Yaskawa INFORM job: FMTV_FENDERS.JBI

/JOB
//NAME FMTV_FENDERS
//POS
///NPOS 545,0,0,3,0,0
///TOOL 0
///POSTYPE PULSE
///PULSE
C00000=-63956,-155148,126845,-105314,-81595,-126672
C00001=-236501,-175042,15743,-102650,-110361,-51662
C00002=-236501,-175042,-85215,-102650,-110361,-73822
C00003=-248122,-122895,-115006,-97112,-80000,-47589
C00004=-248635,-127033,-112745,-102549,-53011,-48741
C00005=-234079,-137705,-95028,-87046,-41878,-79782
C00006=-238942,-134708,-94740,-89961,-45016,-68159
C00007=-242508,-132671,-97164,-92994,-47428,-52176
C00008=-224790,-161630,-99096,-61743,-42779,-71567
C00009=-225833,-166497,-100724,-75197,-37378,-66529
C00010=-225972,-169847,-101473,-88583,-33472,-60957
C00011=-240574,-167077,-99779,-106864,-55530,-59132
C00012=-246383,-162026,-96863,-119993,-73009,-60358
C00013=-241063,-171089,-91582,-115750,-67016,-71356
C00014=-234594,-170823,-91883,-123396,-77107,-68502
C00015=-231990,-170973,-91438,-122280,-75787,-65647
C00016=-218685,-173595,-93676,-116936,-69568,-59454
C00017=-209410,-168993,-95200,-117606,-79816,-56023
C00018=-205376,-166532,-94796,-118730,-93657,-54826
C00019=-205520,-167299,-149545,-118775,-93902,539
C00020=194752,-167299,-149545,-204519,-57378,33957
C00021=227777,-146515,-121429,-211592,-64921,47742
C00022=140813,-165782,-97540,-184911,-23121,3391
C00023=142401,-166246,-97145,-186466,-22763,-397
C00024=129538,-168092,-98000,-174243,-22289,-10940
C00025=108353,-169637,-101483,-151757,-24269,-29279
C00026=76493,-168015,-109892,-143048,-39020,-42938
C00027=71930,-167798,-152447,-142497,-39770,-44912
C00028=-184184,-167798,-152447,-142497,-39770,-44912
C00029=-188241,-175091,-112594,-105313,-81595,-75530
C00030=-137238,-129578,-121502,-201786,-71124,-123955
C00031=-113155,-108086,-93765,-247340,-66179,-146822
C00032=-87884,-87482,-101015,-240031,-88214,-149958
C00033=-87337,-86742,-96838,-237644,-87662,-149095
C00034=-86639,-91328,-99206,-236722,-87486,-148429
C00035=-86780,-92686,-99571,-236735,-87113,-148223
C00036=-87673,-96396,-100101,-236785,-85664,-145021
C00037=-90528,-100864,-97206,-241818,-78899,-142882
C00038=-88930,-100173,-90592,-254807,-82341,-140248
C00039=-88930,-100173,-90592,-254807,-82341,-140248
C00040=-91958,-101268,-92449,-250564,-79276,-141210
C00041=-93563,-102238,-93369,-248531,-77706,-141653
C00042=-119301,-108319,-88132,-240089,-57325,-143963
C00043=-119660,-108541,-87987,-240161,-57013,-143942
C00044=-119839,-108971,-88005,-240265,-56797,-143863
C00045=-120234,-109926,-88726,-240307,-56496,-143882
C00046=-121927,-111036,-90334,-239348,-55531,-144622
C00047=-118976,-116509,-91716,-240930,-60604,-142515
C00048=-116081,-121406,-92670,-241702,-65588,-140629
C00049=-113168,-125880,-93367,-241813,-70447,-138887
C00050=-109736,-130380,-93806,-241238,-75765,-137011
C00051=-105270,-135511,-94001,-239583,-82236,-134673
C00052=-98930,-140934,-93505,-236003,-90100,-131558
C00053=-89867,-146515,-92095,-228369,-100341,-126955
C00054=-89580,-147813,-92127,-228164,-100030,-126621
C00055=-90841,-147991,-91556,-228656,-99205,-126757
C00056=-96418,-152558,-96101,-230948,-96589,-127979
C00057=-91724,-166412,-117528,-260601,-98993,-131473
C00058=-142876,-156018,-103642,-277845,-66892,-131209
C00059=-141572,-151863,-98523,-277546,-67748,-131008
C00060=-143622,-155846,-98171,-279282,-66778,-129574
C00061=-141572,-151863,-98523,-277546,-67748,-131008
C00062=-172590,-143236,-94657,-288827,-48166,-129963
C00063=-191755,-131411,-90127,-295423,-35245,-129238
C00064=-192589,-130434,-90093,-295337,-34548,-129452
C00065=-191324,-128508,-89233,-293789,-35094,-130268
C00066=-170465,-108298,-84931,-276180,-46986,-139791
C00067=-170465,-108298,-84931,-276180,-46986,-139791
C00068=-170175,-107085,-84636,-275676,-47146,-140161
C00069=-170577,-105937,-83925,-275538,-46851,-140322
C00070=-169650,-103921,-80673,-282063,-48979,-138868
C00071=-168642,-102219,-80355,-281188,-49540,-139276
C00072=-169071,-108002,-93409,-278198,-48715,-141830
C00073=-169071,-108002,-93409,-278198,-48715,-141830
C00074=-47220,-130234,-115451,-278198,-65852,-141829
C00075=198695,-175103,-103633,-278198,-100436,-141828
C00076=239511,-167652,-97207,-278198,-100438,-141828
C00077=238443,-174672,23867,-278198,-100438,-141828
C00078=2947,-175103,38446,-278198,-100436,-36834
C00079=16726,-130618,77154,-263150,-91818,-20452
C00080=23551,-123817,76415,-256358,-86647,-25076
C00081=25255,-134753,53984,-254887,-87968,-28104
C00082=34217,-129882,61937,-248584,-86650,-23141
C00083=34992,-129505,62675,-248048,-86512,-23065
C00084=35569,-128900,63365,-247642,-86445,-23063
C00085=35569,-128900,63365,-247642,-86445,-23063
C00086=35569,-128900,63365,-247642,-86445,-23063
C00087=35799,-128709,63623,-247480,-86412,-23052
C00088=36324,-128461,64149,-247118,-86309,-22994
C00089=36692,-142226,36581,-233091,-77214,-27321
C00090=36971,-139485,43358,-233271,-75982,-27198
C00091=42868,-132233,61112,-235070,-77346,-25322
C00092=50739,-147582,43443,-222735,-62053,-31597
C00093=47831,-140548,57273,-230647,-62785,-28767
C00094=34340,-130815,75810,-246275,-65428,-24880
C00095=33507,-162796,67711,-252752,-61051,-17702
C00096=33260,-171150,47504,-183611,-66896,-17832
C00097=100012,-174561,95289,18814,-62607,-57140
C00098=99763,-174577,58172,18619,-63102,-57088
C00099=101096,-171100,56758,19675,-60596,-57340
C00100=84534,-174582,50021,23554,-70995,-76849
C00101=83318,-171811,53916,22816,-71627,-76924
C00102=83719,-170735,55890,22980,-71982,-76759
C00103=84083,-169443,57369,23169,-72011,-76683
C00104=82602,-172191,48669,33395,-63575,-78747
C00105=81200,-174768,38987,47055,-54860,-82592
C00106=83526,-167021,50934,46962,-56546,-75402
C00107=83546,-144153,93765,41175,-74852,-61002
C00108=81875,-142151,96395,45526,-72096,-57806
C00109=83151,-130904,116355,41565,-65822,-44019
C00110=83644,-126633,124240,39180,-65180,-40041
C00111=83534,-127495,122450,39269,-64858,-40238
C00112=84956,-132447,112751,40602,-62697,-40874
C00113=87573,-136499,104656,41438,-60781,-40939
C00114=89464,-137800,101703,41543,-59955,-40657
C00115=90888,-139642,97462,43059,-58642,-40845
C00116=92923,-141988,91755,45353,-56827,-41168
C00117=97347,-145437,82552,50313,-53590,-41778
C00118=101127,-147299,76883,54509,-51347,-42234
C00119=112694,-149561,67089,67207,-46322,-43420
C00120=112404,-142486,73485,67419,-46217,-43743
C00121=112249,-142557,71998,67965,-45978,-44258
C00122=112309,-135857,81532,66813,-46484,-43309
C00123=112423,-127896,93799,65107,-47307,-41879
C00124=112481,-118724,108063,63143,-48368,-40240
C00125=112694,-149561,67089,67207,-46322,-43420
C00126=112694,-149561,67089,67207,-46322,-43420
C00127=116026,-148180,67774,69460,-45423,-43446
C00128=118687,-144460,72072,70778,-44893,-43092
C00129=113027,-132465,87179,66269,-46758,-27490
C00130=113284,-132594,85154,67245,-46318,-28134
C00131=117715,-137204,78104,70883,-44882,-37107
C00132=118231,-136060,79389,71132,-44786,-37034
C00133=118721,-135959,79407,71463,-44662,-37033
C00134=139669,-145382,63973,87795,-39566,-47806
C00135=144694,-152917,52086,93827,-38613,-57145
C00136=151618,-163514,32928,104061,-38168,-72003
C00137=153104,-166256,24026,108879,-38853,-74649
C00138=149828,-162760,31507,104102,-38640,-63057
C00139=147298,-159676,37324,100611,-38673,-54667
C00140=147603,-160409,36248,101031,-38660,-54816
C00141=147925,-161389,34936,101456,-38648,-54956
C00142=148129,-162398,33663,101755,-38646,-55064
C00143=147893,-163417,32335,102136,-38757,-54575
C00144=146258,-164194,31781,100421,-38883,-51526
C00145=140568,-164282,32355,94404,-49003,-49367
C00146=133209,-162489,36110,88716,-64281,-46826
C00147=128857,-160624,39192,86775,-74962,-45374
C00148=126945,-159418,41079,86406,-80510,-44608
C00149=124614,-158041,43286,86500,-87890,-43559
C00150=124939,-153213,57755,86544,-88151,-40924
C00151=125394,-169115,39061,86896,-87980,-41582
C00152=125574,-175038,-5981,87026,-114787,-41677
C00153=125574,-175038,-98531,87026,-114787,-41677
C00154=-224301,-140149,-112569,-110141,-97352,-69368
C00155=-229663,-142484,-108537,-111899,-99628,-71764
C00156=-230892,-138053,-104282,-112208,-100447,-71858
C00157=-228508,-142108,-101165,-112055,-97629,-73428
C00158=-230003,-144530,-99119,-112804,-97681,-74805
C00159=-237315,-146893,-98401,-115581,-101333,-76663
C00160=-237192,-144365,-100145,-122189,-107894,-76884
C00161=-235565,-140992,-101778,-130482,-115488,-77678
C00162=-235563,-141001,-101786,-130481,-115487,-77677
C00163=-237825,-141777,-101649,-131712,-116315,-78485
C00164=-238364,-143167,-100756,-132394,-115806,-79161
C00165=-226999,-153783,-87557,-130027,-102586,-81819
C00166=-222820,-155853,-86813,-128215,-99812,-81611
C00167=-216816,-162804,-92469,-125449,-96634,-80821
C00168=-216816,-162804,-92469,-125449,-96634,-80821
C00169=50184,-164124,-141814,36356,38768,-145446
C00170=54442,-155394,-111475,22539,120746,-180496
C00171=51486,-150306,-107537,20755,122050,-181495
C00172=63426,-151628,-102258,27464,115883,-177940
C00173=71735,-149481,-97078,31867,112002,-175642
C00174=81923,-149105,-93748,36922,107221,-173076
C00175=93853,-150952,-94431,42518,102084,-170079
C00176=97845,-151639,-92939,44162,99620,-169505
C00177=100339,-151371,-92202,45229,98399,-168996
C00178=100309,-151030,-92216,45235,98542,-168932
C00179=100415,-149962,-92546,45356,98998,-168621
C00180=111889,-132617,-94399,56113,85553,-159405
C00181=116128,-123385,-93936,57705,78449,-155514
C00182=119709,-114359,-92766,57352,71837,-151949
C00183=122591,-105709,-90679,55611,66072,-148743
C00184=121430,-103362,-88798,55594,66891,-148891
C00185=120850,-102704,-88701,55530,67390,-148888
C00186=120281,-102346,-88871,55475,67872,-148893
C00187=103719,-103787,-98738,55205,79854,-156387
C00188=103861,-103141,-98570,55164,79915,-156243
C00189=96021,-102003,-100562,55140,85368,-157297
C00190=90958,-101699,-103793,55098,89327,-157636
C00191=89909,-100879,-104523,55097,90388,-157513
C00192=89807,-100027,-104366,55100,90656,-157377
C00193=89221,-98801,-103895,56224,91516,-157316
C00194=88766,-97677,-103297,57173,92190,-157270
C00195=89816,-94344,-102182,57192,92197,-156513
C00196=96964,-101233,-114771,56885,89487,-153707
C00197=96964,-175067,-154909,56885,89487,-153707
C00198=-188147,-175067,-154909,56885,89487,-153707
C00199=-249562,-175082,-16518,56885,115648,-153706
C00200=-188145,-175086,16419,56885,121874,-153706
C00201=-177417,-173959,29423,-34415,105748,-147371
C00202=-215218,-169631,-6124,-67662,97554,-158481
C00203=-212851,-170254,-11358,-66279,98657,-160355
C00204=-199538,-170974,-5542,-56389,98010,-158467
C00205=-196518,-171702,4598,-68884,91761,-156498
C00206=-191507,-170789,17376,-83691,87075,-153205
C00207=-184847,-169628,24159,-91154,83928,-151061
C00208=-184769,-168513,30877,-91403,83962,-149508
C00209=-166653,-153882,67375,-118564,90914,-139805
C00210=-168376,-157673,56992,-119714,89739,-141501
C00211=-170268,-156203,59245,-123438,80532,-141325
C00212=-171412,-154267,62166,-126915,71162,-140836
C00213=-171531,-154006,62478,-127383,69855,-140765
C00214=-172026,-152514,64166,-129774,63219,-140319
C00215=-172277,-150476,66358,-132476,56004,-139609
C00216=-172404,-145153,73532,-132977,56608,-139199
C00217=-171743,-142696,76210,-132662,56537,-139081
C00218=-175468,-149312,61635,-117570,52509,-146387
C00219=-182053,-156892,41178,-91409,54589,-159429
C00220=-179598,-153809,48467,-91200,54250,-158022
C00221=-177876,-151695,51361,-90271,53969,-157773
C00222=-175031,-149700,54466,-88701,53470,-157416
C00223=-171138,-149200,55226,-90700,51887,-155676
C00224=-152905,-141663,70200,-105827,48301,-143509
C00225=-152337,-141979,69626,-105360,48147,-143575
C00226=-151943,-142781,68394,-104935,48012,-143705
C00227=-148029,-134110,86517,-121166,52616,-135065
C00228=-146834,-130705,93327,-125465,54888,-132704
C00229=-145103,-124844,104734,-130953,58789,-129572
C00230=-142768,-113260,126814,-137507,65892,-125434
C00231=-135917,-118098,122435,-150990,58780,-120039
C00232=-136643,-115604,126770,-151681,59833,-118172
C00233=-133945,-127048,108732,-147879,54997,-122652
C00234=-132685,-131473,101421,-146007,52903,-123186
C00235=-131275,-135352,94587,-143913,50769,-123796
C00236=-131275,-135352,94587,-143913,50769,-123796
C00237=-131275,-135352,94587,-143913,50769,-123796
C00238=-121206,-145281,78428,-130981,41887,-126182
C00239=-108596,-150086,71319,-118128,35191,-127801
C00240=-108596,-150086,71319,-118128,35191,-127801
C00241=-108596,-150086,71319,-118128,35191,-127801
C00242=-106173,-149311,73486,-117873,34909,-126912
C00243=-105014,-148827,74616,-117745,34762,-126490
C00244=-103301,-148028,76337,-117552,34523,-125880
C00245=-101267,-148049,76425,-114785,33084,-126447
C00246=-98887,-147633,77014,-111606,31465,-127110
C00247=-99861,-135336,105011,-122576,35238,-120303
C00248=-79582,-141041,101392,-54417,-60770,-149548
C00249=-78156,-144611,92640,-54931,-59723,-148027
C00250=-76477,-145690,87146,-55172,-58933,-146653
C00251=-76325,-152698,75551,-53287,-65768,-134624
C00252=-76716,-159478,64431,-47040,-68901,-125086
C00253=-79518,-161789,63221,-35636,-69401,-124582
C00254=-81209,-163290,61958,-29327,-69264,-124632
C00255=-84722,-166411,58236,-19438,-67363,-126288
C00256=-86671,-168300,55657,-13814,-66439,-127558
C00257=-86671,-168300,55657,-13814,-66439,-127558
C00258=-86216,-169741,53857,-13592,-66313,-127456
C00259=-85119,-170597,52676,-13583,-66937,-127129
C00260=-82515,-161498,64875,-12910,-80387,-133971
C00261=-77611,-145974,86579,-16344,-98063,-141066
C00262=-78076,-150431,78979,-16594,-96561,-139590
C00263=-80411,-152118,77648,-18159,-96529,-140021
C00264=-82668,-153005,77611,-19681,-96705,-140485
C00265=-88888,-175086,79531,-19379,-96436,-140350
C00266=-110968,-175086,9069,-19379,-125140,-140350
C00267=-110968,-175086,-114864,-19379,-125140,-140350
C00268=175304,-175086,-114864,-19379,-30472,-99694
C00269=187329,-129396,-122749,-38461,29346,-63021
C00270=183916,-109052,-100373,-57748,65750,-30233
C00271=197239,-90135,-82008,-58535,73988,-27553
C00272=201754,-94869,-83954,-58993,75937,-25896
C00273=202079,-95139,-84115,-59008,76103,-25800
C00274=202637,-95511,-84460,-59016,76432,-25674
C00275=202637,-95511,-84460,-59016,76432,-25674
C00276=202637,-95511,-84460,-59016,76432,-25674
C00277=202860,-95637,-84608,-59016,76571,-25633
C00278=203690,-96180,-85102,-59023,77053,-25445
C00279=208915,-99439,-88258,-58000,79285,-28016
C00280=205478,-105010,-93814,-58035,77197,-28705
C00281=214139,-97501,-89593,-72382,81942,-36081
C00282=224242,-84526,-78845,-86787,78269,-51115
C00283=224432,-83745,-74911,-87107,78310,-50227
C00284=223676,-86642,-76315,-87324,77734,-49801
C00285=223812,-88001,-76982,-87395,77808,-49593
C00286=224543,-88686,-77346,-87375,78313,-49481
C00287=235420,-107309,-83637,-91467,63449,-46681
C00288=240320,-114099,-85995,-93455,57854,-45609
C00289=246996,-121668,-88445,-96053,51244,-44273
C00290=246996,-121668,-88445,-96053,51244,-44273
C00291=249717,-122652,-88778,-95572,53097,-44156
C00292=250120,-123785,-89127,-95767,53405,-43893
C00293=232812,-141826,-96443,-115069,24978,-36767
C00294=232812,-141826,-96443,-115069,24978,-36767
C00295=233391,-143923,-96937,-116153,25668,-36002
C00296=237215,-145543,-97234,-114188,28169,-36484
C00297=245415,-146262,-97619,-108727,33105,-38331
C00298=245415,-146262,-97619,-108727,33105,-38331
C00299=247668,-147105,-97798,-107850,34572,-38441
C00300=248141,-148229,-98044,-108198,34996,-38104
C00301=248169,-149917,-101541,-106958,34753,-38928
C00302=248344,-161240,-125557,-97827,33569,-44956
C00303=179896,-161240,-125557,-97827,-77291,-48113
C00304=184979,-139013,-125331,-99817,-75478,-48047
C00305=179112,-130483,-99577,-98597,-78190,-53181
C00306=178361,-129263,-96461,-98549,-78560,-53744
C00307=161550,-139106,-101847,-102031,-89241,-56097
C00308=150835,-139809,-97057,-95903,-96892,-60596
C00309=132439,-136388,-86127,-87364,-112558,-64828
C00310=125150,-133069,-79774,-83061,-119517,-65455
C00311=123583,-134542,-82111,-83279,-120436,-65117
C00312=123583,-134540,-118710,-83279,-120438,-65115
C00313=-136821,-161457,-114880,15988,-123554,-94299
C00314=-194311,-175100,-121530,66302,-125133,-109092
C00315=-194311,-175100,-121530,-44006,100681,-109092
C00316=-254343,-175097,-89612,-83602,114959,-15902
C00317=-134289,-173861,-75426,-80327,116995,-14503
C00318=-122808,-169798,-71461,-73331,121943,-13820
C00319=-204100,-166260,-61655,-119208,88598,-10349
C00320=-223955,-164817,-61952,-125089,83393,-8296
C00321=-234599,-164424,-61970,-128682,80581,-6975
C00322=-239551,-164319,-62025,-130691,79207,-6317
C00323=-239846,-164373,-60068,-133976,79268,-5541
C00324=-241352,-164565,-58325,-139265,78932,-4470
C00325=-241352,-164565,-58325,-139265,78932,-4470
C00326=-241352,-164565,-58325,-139265,78932,-4470
C00327=-247260,-164414,-57679,-143144,77614,-3349
C00328=-250453,-164099,-56779,-145288,77091,-2673
C00329=-231804,-169514,-49324,-147051,71343,-6571
C00330=-232933,-169740,-48497,-147965,71587,-6225
C00331=-232886,-175090,-53650,-147961,71735,-6180
C00332=-241976,-170697,-124750,-139782,79456,-4031
C00333=-176745,-151691,-107508,-102764,25310,-35154
C00334=-176745,-151691,-107508,-102764,25310,-35154
C00335=-175824,-150531,-104417,-104152,26105,-34141
C00336=-176745,-151691,-107508,-102764,25310,-35154
C00337=-195718,-137133,-102300,-100933,12070,-39089
C00338=-195586,-136734,-99661,-105865,12408,-36294
C00339=-195718,-137133,-102300,-100933,12070,-39089
C00340=-180125,-124233,-99711,-80430,22769,-49034
C00341=-179992,-123952,-97169,-83121,22691,-47416
C00342=-180125,-124233,-99711,-80430,22769,-49034
C00343=-162775,-136432,-106392,-85396,34185,-43914
C00344=-162116,-135482,-103340,-86834,34551,-42863
C00345=-162775,-136432,-106392,-85396,34185,-43914
C00346=-136686,-149350,-103002,-109734,61122,-29919
C00347=-106697,-140430,-78975,-133534,56483,-36128
C00348=-113088,-137327,-73738,-138383,54551,-33834
C00349=-113904,-135440,-73782,-138477,53489,-34041
C00350=-109003,-138587,-73014,-136035,56934,-34530
C00351=-120827,-140923,-75250,-144601,52532,-30939
C00352=-120374,-136814,-75228,-143259,51004,-31973
C00353=-120840,-133958,-75226,-142869,49667,-32458
C00354=-120840,-133958,-75226,-142869,49667,-32458
C00355=-118039,-132206,-74509,-140437,50317,-33657
C00356=-114795,-132712,-73740,-138398,52103,-34407
C00357=-113063,-135707,-73613,-137984,53990,-34190
C00358=-109736,-137390,-76478,-135398,54956,-35431
C00359=-89018,-147818,-96006,-121054,62352,-42706
C00360=-127918,-122489,-87741,-140529,17400,-4354
C00361=-127917,-122488,-87741,-140529,17399,-4355
C00362=-120737,-122510,-87236,-129675,21028,-9702
C00363=-118823,-120927,-84702,-128126,22316,-10351
C00364=-119175,-120684,-84537,-128485,22104,-10188
C00365=-118541,-120339,-84470,-127414,22352,-10732
C00366=-117917,-120545,-84643,-126699,22698,-11070
C00367=-117746,-121573,-84792,-127367,23061,-10647
C00368=-117746,-121573,-84792,-127367,23061,-10647
C00369=-118346,-121848,-84823,-128327,22818,-10162
C00370=-118860,-121524,-84661,-128795,22499,-9956
C00371=-119121,-120634,-84551,-128353,22112,-10259
C00372=-120130,-121883,-86413,-129062,21401,-9982
C00373=-136794,-118620,-79645,-163280,16358,7465
C00374=-138097,-118087,-78864,-166565,16237,9158
C00375=-135793,-117588,-77729,-161369,16975,6516
C00376=-135907,-117348,-77360,-161699,17008,6690
C00377=-135907,-117348,-77360,-161699,17008,6690
C00378=-135643,-117215,-77441,-160973,16962,6311
C00379=-135311,-117474,-77621,-160262,17078,5951
C00380=-135426,-118271,-77715,-160928,17394,6320
C00381=-135426,-118271,-77715,-160928,17394,6320
C00382=-135616,-118450,-77670,-161479,17461,6609
C00383=-135939,-118199,-77498,-162164,17351,6954
C00384=-135907,-117348,-77360,-161699,17008,6690
C00385=-136699,-118602,-79632,-163041,16374,7342
C00386=-136699,-118602,-79632,-163041,16374,7342
C00387=-165437,-150621,-99310,-185487,43820,-1784
C00388=-239107,-166921,-73717,-195647,87109,-7095
C00389=-194457,-169656,-47982,-122093,99629,-6955
C00390=-192738,-162336,-43403,-121261,99351,-7823
C00391=-189653,-162700,-44245,-119457,100137,-8226
C00392=-184748,-163106,-42837,-116371,102013,-8193
C00393=-185120,-162960,-40552,-116390,102376,-7617
C00394=-187523,-162625,-39967,-117823,101744,-7357
C00395=-189522,-162401,-40080,-119065,101109,-7283
C00396=-196021,-161852,-41671,-123148,98752,-7201
C00397=-196021,-161852,-41671,-123148,98752,-7201
C00398=-205203,-161164,-42254,-128753,95884,-6511
C00399=-201648,-161772,-46731,-126775,95696,-7779
C00400=-190472,-162626,-44480,-119970,99820,-8220
C00401=-190313,-162622,-44069,-119843,99965,-8142
C00402=-192361,-162380,-43509,-121042,99444,-7873
C00403=-194583,-165726,-46201,-122322,99000,-7481
C00404=-151983,-172688,-34997,-92919,112988,-4614
C00405=-149743,-170439,-33113,-91511,113496,-4751
C00406=-148403,-170692,-30265,-89926,113802,-3812
C00407=-150361,-170138,-28085,-90907,113399,-3327
C00408=-152728,-169497,-28204,-92676,112905,-3554
C00409=-154075,-169277,-30854,-94182,112537,-4403
C00410=-154075,-169277,-30854,-94182,112537,-4403
C00411=-158038,-168535,-32458,-97285,111515,-5058
C00412=-153030,-169970,-36759,-94565,112608,-5968
C00413=-149954,-170620,-32630,-91507,113456,-4549
C00414=-151149,-170283,-32638,-92384,113180,-4650
C00415=-152677,-172683,-34781,-93339,112839,-4546
C00416=-152677,-172683,-34781,-93339,112839,-4546
C00417=-202662,-172683,11619,-93339,112839,48019
C00418=-172079,-162006,55824,-105048,97973,50689
C00419=-156965,-147756,77669,-110835,90627,52009
C00420=-162605,-134946,89084,-112919,91170,61307
C00421=-163977,-138528,79786,-113850,90417,59792
C00422=-163864,-138373,79921,-113775,90385,59791
C00423=-163868,-138296,80030,-113777,90392,59798
C00424=-163718,-138715,79353,-113677,90308,59744
C00425=-163827,-138924,79143,-113750,90334,59739
C00426=-164442,-138353,80353,-114158,90602,59864
C00427=-164442,-138353,80353,-114158,90602,59864
C00428=-164540,-138058,80828,-114223,90661,59902
C00429=-164383,-137873,80971,-114119,90616,59899
C00430=-163868,-138296,80030,-113777,90392,59798
C00431=-163745,-138241,80515,-113696,90449,59913
C00432=-163403,-136976,83718,-113464,90741,60418
C00433=-161326,-138645,80849,-112099,90007,60237
C00434=-161945,-140167,76597,-112502,89652,59512
C00435=-162084,-140314,76484,-112595,89692,59513
C00436=-162084,-140314,76484,-112595,89692,59513
C00437=-162240,-139895,77149,-112701,89773,59565
C00438=-162118,-139700,77337,-112620,89743,59569
C00439=-161618,-140063,76526,-112286,89547,59483
C00440=-161618,-140063,76526,-112286,89547,59483
C00441=-161417,-140517,75787,-112151,89449,59423
C00442=-161560,-140745,75567,-112246,89484,59419
C00443=-162084,-140314,76484,-112595,89692,59513
C00444=-162099,-140035,76871,-112605,89714,59538
C00445=-160829,-134754,90109,-111762,90847,61622
C00446=-159720,-161570,51808,-110997,88636,58885
C00447=-159720,-161570,51808,-110997,88636,58885
C00448=-66393,-161570,77783,-97808,-20643,67154
C00449=-1098,-161570,51808,-88581,-112832,48915
C00450=-816,-175088,-83121,-88456,-117207,57832
C00451=66284,-151327,-103203,-82579,-59616,118766
C00452=125030,-126740,-90074,-53431,-21483,109123
C00453=122149,-124544,-86727,-55767,-23360,110091
C00454=122152,-124880,-86870,-55572,-23415,109973
C00455=122152,-124880,-86870,-55572,-23415,109973
C00456=121786,-125023,-86853,-55823,-23665,110073
C00457=121410,-124848,-86884,-56435,-23810,110383
C00458=121508,-123953,-86775,-57108,-23530,110801
C00459=121508,-123953,-86775,-57108,-23530,110801
C00460=122083,-123590,-86609,-56673,-23154,110628
C00461=122274,-124059,-86747,-56125,-23145,110328
C00462=122152,-124880,-86870,-55572,-23415,109973
C00463=121928,-124654,-86798,-55974,-23492,110182
C00464=124210,-126123,-89128,-54129,-22015,109417
C00465=141312,-121381,-81155,-20494,-16221,92438
C00466=138752,-120051,-78743,-25647,-17363,95006
C00467=139021,-120477,-78695,-24731,-17508,94522
C00468=139021,-120477,-78695,-24731,-17508,94522
C00469=138791,-120658,-78818,-25184,-17599,94748
C00470=138539,-120594,-78914,-25836,-17597,95084
C00471=138387,-119804,-78859,-26699,-17303,95557
C00472=138387,-119804,-78859,-26699,-17303,95557
C00473=138747,-119437,-78647,-26033,-17125,95228
C00474=139019,-119675,-78568,-25205,-17193,94793
C00475=139021,-120477,-78695,-24731,-17508,94522
C00476=138801,-120508,-78792,-25251,-17539,94787
C00477=141556,-122106,-82352,-20173,-15951,92291
C00478=135806,-142290,-83979,-21960,-26197,92274
C00479=66284,-151327,-103203,-82579,-59616,118766
C00480=-1098,-173731,-82817,-88581,-117340,57859
C00481=-1098,-161570,51808,-88581,-112832,48915
C00482=84231,-163436,65647,-87836,-97055,57895
C00483=163264,-143645,78465,-87146,-97014,43961
C00484=163460,-129192,97130,-69494,-94201,37055
C00485=164010,-131942,90570,-69017,-93676,38056
C00486=163856,-132419,89787,-69109,-93584,38124
C00487=163856,-132419,89787,-69109,-93584,38124
C00488=163664,-132234,89921,-69235,-93522,38127
C00489=163827,-131810,90631,-69134,-93615,38065
C00490=164281,-131423,91490,-68853,-93818,37971
C00491=164281,-131423,91490,-68853,-93818,37971
C00492=164440,-131498,91495,-68750,-93874,37958
C00493=164322,-131924,90804,-68821,-93797,38016
C00494=163856,-132419,89787,-69109,-93584,38124
C00495=163938,-132086,90314,-69061,-93639,38080
C00496=163490,-129894,95565,-69446,-94061,37276
C00497=165665,-127416,100500,-68114,-95112,36796
C00498=166116,-129701,95149,-67704,-94662,37598
C00499=166026,-130145,94439,-67754,-94589,37658
C00500=166026,-130145,94439,-67754,-94589,37658
C00501=165874,-130012,94518,-67853,-94540,37663
C00502=166012,-129462,95418,-67775,-94641,37584
C00503=166510,-128915,96591,-67472,-94896,37461
C00504=166510,-128915,96591,-67472,-94896,37461
C00505=166609,-129059,96459,-67407,-94928,37464
C00506=166512,-129578,95631,-67458,-94845,37533
C00507=166026,-130145,94439,-67754,-94589,37658
C00508=166032,-129926,94759,-67754,-94609,37633
C00509=165482,-127109,101350,-68255,-95161,36645
C00510=164208,-159322,58583,-68782,-93006,39082
C00511=164208,-159322,58583,-68782,-93006,39082
C00512=224736,-167682,40736,-68782,-105264,72730
C00513=194680,-164791,-39980,-51259,-102330,-91617
C00514=191540,-160851,-36926,-53053,-102784,-91063
C00515=184807,-161527,-34772,-57388,-105265,-91064
C00516=185201,-161205,-32929,-57325,-105583,-91467
C00517=189291,-160565,-32118,-54852,-104661,-91878
C00518=194463,-160090,-33718,-51511,-102836,-91912
C00519=194463,-160090,-33718,-51511,-102836,-91912
C00520=202965,-159248,-35158,-46209,-100147,-92377
C00521=196802,-160399,-39171,-49701,-100634,-91054
C00522=190344,-161045,-36414,-53830,-103291,-91100
C00523=191696,-160773,-35801,-53050,-103062,-91316
C00524=194174,-164245,-38599,-51627,-102708,-91745
C00525=194174,-164245,-38599,-51627,-102708,-91745
C00526=198339,-174688,-65015,-37413,-79325,-95361
C00527=204067,-174898,-119878,7219,-14454,-108471
C00528=198954,-152362,-105597,-9824,-10053,-99837
C00529=197427,-150836,-102190,-14366,-11165,-97559
C00530=198954,-152362,-105597,-9824,-10053,-99837
C00531=179244,-139699,-104769,-78536,-15484,-64306
C00532=177962,-138324,-101526,-76366,-16523,-65725
C00533=179244,-139699,-104769,-78536,-15484,-64306
C00534=195169,-125451,-98204,-94015,-4294,-53834
C00535=194122,-124841,-95314,-80722,-5075,-61281
C00536=195169,-125451,-98204,-94015,-4294,-53834
C00537=213212,-135016,-100603,-103392,8077,-46604
C00538=212592,-134163,-97665,-111459,7983,-42204
C00539=213212,-135016,-100603,-103392,8077,-46604
C00540=254380,-167483,-141973,-103392,-66077,-46604
C00541=254380,-175085,6002,-103392,-92921,-46604
C00542=48314,-162179,62962,-104636,-85589,-98434
C00543=7562,-158757,35528,-104747,-84933,-103069
C00544=-63956,-155148,126845,-105314,-81595,-126672
///POSTYPE TOOL
///RECTAN
///RCONF 0,0,0,0,0,0,0,0,0,0,0,0,0,0,0,0,0,0,0,0,0,0,0,0
P00101=-6.500,-0.500,8.000,0.0000,0.0000,0.0000
P00102=-7.000,0.000,3.000,0.0000,0.0000,0.0000
P00103=0.500,1.750,0.000,0.0000,0.0000,0.0000
//INST
///DATE 2023/09/19 13:13
///ATTR SC,RW
///GROUP1 RB1
NOP
CALL JOB:SYS_SPINDLE_START
CALL JOB:SYS_FILTERS_START
CALL JOB:SYS_GATE_LOCK
CALL JOB:SYS_VERIFY_GATE_LOCKED
MOVJ C00000 VJ=15.42  //HOME
MOVJ C00001 VJ=15.42  //ABOVE
MOVJ C00002 VJ=20.56  //ABOVE
CALL JOB:EARCUT
MOVJ C00003 VJ=20.56  //ABOVE
MOVJ C00004 VJ=20.56  //ABOVE
MOVL C00005 V=50.0  //INTO
MOVL C00006 V=6.3
MOVL C00007 V=6.3  //1ST FLASH
MOVL C00008 V=6.3  //2ND
MOVL C00009 V=6.3
MOVL C00010 V=6.3
MOVL C00011 V=6.3
MOVL C00012 V=6.3
MOVL C00013 V=6.3
MOVL C00014 V=6.3
MOVL C00015 V=6.3
MOVL C00016 V=6.3
MOVL C00017 V=6.3
MOVL C00018 V=6.3  //END FLASH
MOVJ C00019 VJ=27.42  //ABOVE
MOVJ C00020 VJ=27.42  //ROTATE
MOVL C00021 V=50.0  //INLINE 2ND FLASH
MOVL C00022 V=6.3  //1ST CORNER
MOVL C00023 V=6.3  //2ND
MOVL C00024 V=6.3
MOVL C00025 V=6.3
MOVL C00026 V=15.0  //OUT 2ND FLASH
MOVJ C00027 VJ=50.00
MOVJ C00028 VJ=50.00  //RIGHT
MOVJ C00029 VJ=50.00  //OVER RIGHT FENDER
MOVJ C00030 VJ=50.00
MOVJ C00031 VJ=50.00
MOVL C00032 V=150.0  //UP TO FRONT CUT
MOVL C00033 V=100.0  //INLINE
MOVC C00034 V=6.3  //INTO
MOVC C00035 V=6.3
MOVC C00036 V=6.3
MOVL C00037 V=6.3
MOVL C00038 V=6.3
MOVL C00039 V=4.2
MOVL C00040 V=6.3
MOVL C00041 V=6.3
MOVL C00042 V=6.3
MOVL C00043 V=6.3
MOVL C00044 V=6.3
MOVL C00045 V=6.3
MOVL C00046 V=6.3  //TOP VERTICAL
MOVL C00047 V=6.3
MOVL C00048 V=6.3
MOVL C00049 V=6.3
MOVL C00050 V=6.3
MOVL C00051 V=6.3
MOVL C00052 V=6.3
MOVC C00053 V=6.3
MOVC C00054 V=6.3
MOVC C00055 V=6.3
MOVL C00056 V=18.9  //OUT
MOVJ C00057 VJ=27.42
MOVL C00058 V=150.0  //UP TO
MOVL C00059 V=6.3 PL=0  //INTO TOP CORNER
MOVL C00060 V=6.3 PL=0
MOVL C00061 V=6.3  //INTO TOP CORNER
MOVL C00062 V=6.3
MOVC C00063 V=6.3  //BACK CURVE
MOVC C00064 V=6.3
MOVC C00065 V=6.3
MOVL C00066 V=6.3
MOVC C00067 V=6.3
MOVC C00068 V=6.3
MOVC C00069 V=6.3
MOVL C00070 V=6.3  //BACK STRAIGHT
MOVL C00071 V=6.3
MOVL C00072 V=18.9  //OUT
MOVJ C00073 VJ=50.00
MOVJ C00074 VJ=50.00
MOVJ C00075 VJ=50.00
MOVJ C00076 VJ=50.00 PL=0
MOVJ C00077 VJ=50.00 PL=0
MOVJ C00078 VJ=50.00 PL=0  //ROTATE TO BACK
MOVL C00079 V=150.0
MOVL C00080 V=150.0 PL=0  //UP TO INLINE
MOVL C00081 V=6.3  //INTO BACK
MOVC C00082 V=6.3
MOVC C00083 V=6.3
MOVC C00084 V=6.3
MOVL C00085 V=6.3
MOVC C00086 V=6.3
MOVC C00087 V=6.3
MOVC C00088 V=6.3
MOVL C00089 V=6.3
MOVL C00090 V=6.3
MOVL C00091 V=6.3
MOVL C00092 V=6.3
MOVL C00093 V=6.3  //OUT
MOVL C00094 V=100.0  //AWAY
MOVL C00095 V=150.0  //ABOVE AWAY
MOVJ C00096 VJ=50.00
MOVJ C00097 VJ=50.00
MOVJ C00098 VJ=50.00
MOVL C00099 V=100.0  //ROTATE TO SIDE
MOVL C00100 V=100.0 PL=0  //UP TO
MOVC C00101 V=6.3
MOVC C00102 V=6.3
MOVC C00103 V=6.3
MOVL C00104 V=6.3
MOVL C00105 V=6.3
MOVL C00106 V=6.3
MOVL C00107 V=6.3 PL=0
MOVL C00108 V=6.3 PL=0
MOVL C00109 V=6.3
MOVL C00110 V=6.3
MOVC C00111 V=6.3
MOVC C00112 V=6.3
MOVC C00113 V=6.3
MOVC C00114 V=6.3
MOVC C00115 V=6.3
MOVL C00116 V=6.3
MOVL C00117 V=6.3
MOVL C00118 V=6.3
MOVL C00119 V=6.3
'RELIEF CUT
MOVL C00120 V=6.3
MOVL C00121 V=6.3
MOVL C00122 V=6.3
MOVL C00123 V=6.3
MOVL C00124 V=6.3 PL=0
MOVL C00125 V=6.3 PL=0
MOVC C00126 V=6.3
MOVC C00127 V=6.3
MOVC C00128 V=6.3
MOVL C00129 V=6.3
MOVL C00130 V=6.3
MOVC C00131 V=6.3
MOVC C00132 V=6.3
MOVC C00133 V=6.3
MOVL C00134 V=6.3
MOVL C00135 V=6.3
MOVL C00136 V=6.3
MOVL C00137 V=6.3
MOVL C00138 V=6.3
MOVC C00139 V=6.3
MOVC C00140 V=6.3
MOVC C00141 V=6.3
MOVC C00142 V=6.3
MOVC C00143 V=6.3
MOVC C00144 V=6.3
MOVL C00145 V=6.3
MOVL C00146 V=6.3
MOVL C00147 V=6.3
MOVL C00148 V=6.3
MOVL C00149 V=6.3 PL=0
MOVL C00150 V=18.9  //OUT
MOVL C00151 V=150.0
MOVJ C00152 VJ=50.00
MOVJ C00153 VJ=50.00
MOVJ C00154 VJ=50.00  //ROTATE ABOVE
MOVL C00155 V=50.0  //INLINE
MOVL C00156 V=6.3  //INTO TOP CORNER
MOVC C00157 V=6.3
MOVC C00158 V=6.3
MOVC C00159 V=6.3
MOVL C00160 V=6.3
MOVL C00161 V=6.3
MOVC C00162 V=6.3
MOVC C00163 V=6.3
MOVC C00164 V=6.3
MOVL C00165 V=6.3
MOVL C00166 V=6.3
MOVL C00167 V=18.9  //OUT
MOVJ C00168 VJ=50.00
MOVJ C00169 VJ=50.00
MOVL C00170 V=150.0  //ABOVE LEFT
MOVL C00171 V=100.0  //UP TO
MOVL C00172 V=4.4  //4
MOVL C00173 V=4.4  //3
MOVL C00174 V=4.4  //2
MOVL C00175 V=4.4  //1
MOVL C00176 V=4.4
MOVC C00177 V=4.4
MOVC C00178 V=6.3
MOVC C00179 V=6.3
MOVL C00180 V=11.2
MOVL C00181 V=11.2
MOVL C00182 V=11.2
MOVL C00183 V=11.2
MOVC C00184 V=11.2
MOVC C00185 V=11.2
MOVC C00186 V=11.2
MOVL C00187 V=11.2
MOVL C00188 V=11.2
MOVL C00189 V=11.2
MOVC C00190 V=11.2
MOVC C00191 V=11.2
MOVC C00192 V=11.2
MOVC C00193 V=11.2
MOVC C00194 V=11.2
MOVL C00195 V=11.2  //OUT
MOVL C00196 V=65.0  //AWAY
MOVJ C00197 VJ=48.75  //READY TO ROTATE
MOVJ C00198 VJ=48.75  //ROTATE
MOVJ C00199 VJ=41.25
MOVJ C00200 VJ=48.75  //SWING
MOVJ C00201 VJ=48.75
MOVJ C00202 VJ=41.25
MOVL C00203 V=65.0
MOVL C00204 V=11.2
MOVL C00205 V=11.2
MOVL C00206 V=11.2
MOVL C00207 V=11.2
MOVL C00208 V=33.7  //OUT
MOVL C00209 V=65.0  //INLINE
MOVL C00210 V=11.2  //INTO
MOVL C00211 V=11.2
MOVL C00212 V=11.2
MOVL C00213 V=11.2
MOVL C00214 V=11.2
MOVC C00215 V=11.2
MOVC C00216 V=11.2
MOVC C00217 V=11.2
MOVL C00218 V=11.2
MOVL C00219 V=11.2
MOVC C00220 V=11.2
MOVC C00221 V=11.2
MOVC C00222 V=11.2
MOVL C00223 V=11.2
MOVC C00224 V=11.2
MOVC C00225 V=11.2
MOVC C00226 V=11.2
MOVL C00227 V=11.2
MOVL C00228 V=11.2
MOVL C00229 V=11.2
MOVL C00230 V=11.2
MOVL C00231 V=11.2
MOVC C00232 V=11.2
MOVC C00233 V=11.2
MOVC C00234 V=11.2
MOVC C00235 V=11.2
MOVL C00236 V=11.2
MOVC C00237 V=11.2
MOVC C00238 V=11.2
MOVC C00239 V=11.2
MOVL C00240 V=11.2
MOVC C00241 V=11.2
MOVC C00242 V=11.2
MOVC C00243 V=11.2
MOVC C00244 V=11.2
MOVC C00245 V=11.2
MOVC C00246 V=11.2
MOVL C00247 V=33.7  //OUT
MOVJ C00248 VJ=48.75
MOVL C00249 V=65.0  //UP TO
MOVL C00250 V=11.2  //INTO
MOVL C00251 V=11.2
MOVL C00252 V=11.2  //TOP ROTATING
MOVL C00253 V=11.2
MOVL C00254 V=11.2  //MIDDLE
MOVL C00255 V=11.2
MOVL C00256 V=11.2  //TOP
MOVC C00257 V=11.2
MOVC C00258 V=11.2
MOVC C00259 V=11.2
MOVL C00260 V=11.2
MOVL C00261 V=11.2
MOVL C00262 V=11.2
MOVL C00263 V=33.7  //OUT
MOVJ C00264 VJ=48.75
MOVJ C00265 VJ=48.75
MOVJ C00266 VJ=48.75
MOVJ C00267 VJ=48.75  //ABOVE
MOVJ C00268 VJ=48.75
MOVJ C00269 VJ=48.75
MOVL C00270 V=150.0
MOVL C00271 V=65.0  //UP TO
MOVC C00272 V=11.2
MOVC C00273 V=11.2
MOVC C00274 V=11.2
MOVL C00275 V=11.2
MOVC C00276 V=11.2
MOVC C00277 V=11.2
MOVC C00278 V=11.2
MOVL C00279 V=11.2  //END
MOVL C00280 V=11.2  //OUT
MOVL C00281 V=120.0 PL=0
MOVL C00282 V=120.0 PL=0  //UP TO
MOVL C00283 V=11.2  //INTO
MOVC C00284 V=11.2
MOVC C00285 V=11.2
MOVC C00286 V=11.2
MOVL C00287 V=11.2
MOVL C00288 V=11.2
MOVL C00289 V=11.2
MOVC C00290 V=11.2
MOVC C00291 V=11.2
MOVC C00292 V=11.2
MOVL C00293 V=11.2
MOVC C00294 V=11.2
MOVC C00295 V=11.2
MOVC C00296 V=11.2
MOVL C00297 V=11.2
MOVC C00298 V=11.2
MOVC C00299 V=11.2
MOVC C00300 V=11.2
MOVL C00301 V=33.7
MOVL C00302 V=120.0  //AWAY
MOVL C00303 V=120.0
MOVL C00304 V=120.0  //ABOVE
MOVL C00305 V=120.0  //UP TO
MOVL C00306 V=11.2  //IN
MOVL C00307 V=11.2  //TOP
MOVL C00308 V=11.2
MOVL C00309 V=11.2
MOVL C00310 V=11.2
MOVL C00311 V=33.7  //OUT
MOVJ C00312 VJ=48.75
MOVJ C00313 VJ=48.75
MOVJ C00314 VJ=48.75
MOVJ C00315 VJ=48.75  //ROTATE
MOVJ C00316 VJ=41.25
MOVJ C00317 VJ=18.75  //ABOVE
MOVL C00318 V=11.2  //INTO
MOVC C00319 V=11.2
MOVC C00320 V=11.2
MOVC C00321 V=11.2
MOVC C00322 V=11.2
MOVC C00323 V=11.2
MOVC C00324 V=11.2
MOVL C00325 V=11.2
MOVC C00326 V=11.2
MOVC C00327 V=11.2
MOVC C00328 V=11.2
MOVL C00329 V=11.2
MOVL C00330 V=11.2
MOVL C00331 V=11.2  //OUT
MOVJ C00332 VJ=41.25
COMM CALL JOB:SYS_SPINDLE_STOP
COMM CALL JOB:SYS_UNLOCK_GATE
COMM PAUSE
COMM CALL JOB:SYS_GATE_LOCK
COMM CALL JOB:SYS_VERIFY_GATE_LOCKED
COMM CALL JOB:SYS_SPINDLE_START
COMM TIMER T=8.00
MOVJ C00333 VJ=48.75
MOVL C00334 V=65.0  //UP TO FIRST
MOVL C00335 V=11.2  //INTO FIRST TOP
FORMCUT FCF#(1)
MOVL C00336 V=33.7  //OUT OF 1
MOVL C00337 V=65.0  //UP TO 2
MOVL C00338 V=11.2  //INTO 2ND
FORMCUT FCF#(1)
MOVL C00339 V=33.7  //OUT OF 2
MOVL C00340 V=65.0  //UP TO 3
MOVL C00341 V=11.2  //INTO 3
FORMCUT FCF#(1)
MOVL C00342 V=33.7  //OUT OF 3
MOVL C00343 V=65.0  //UP TO 4
MOVL C00344 V=11.2  //INTO 4
FORMCUT FCF#(1)
MOVL C00345 V=33.7  //OUT OF 4
MOVL C00346 V=65.0  //ABOVE CORNER
MOVL C00347 V=65.0  //ABOVE 1
MOVL C00348 V=11.2  //INTO 1
MOVC C00349 V=11.2
MOVC C00350 V=11.2
MOVC C00351 V=11.2
MOVC C00352 V=11.2
MOVL C00353 V=11.2
MOVC C00354 V=11.2
MOVC C00355 V=11.2
MOVC C00356 V=11.2
MOVL C00357 V=11.2
MOVL C00358 V=33.7  //OUT OF 1
MOVJ C00359 VJ=48.75
MOVJ C00360 VJ=48.75
MOVC C00361 V=15.0
SFTON P101
MOVL C00362 V=65.0  //UP TO 1ST OB
MOVL C00363 V=11.2  //INTO 1ST OB
MOVC C00364 V=11.2
MOVC C00365 V=11.2
MOVC C00366 V=11.2
MOVL C00367 V=11.2
MOVC C00368 V=11.2
MOVC C00369 V=11.2
MOVC C00370 V=11.2
MOVL C00371 V=11.2  //END
SFTOF
MOVL C00372 V=33.7  //OUT
MOVL C00373 V=65.0  //UP TO 2ND OB
MOVL C00374 V=65.0
SFTON P101
MOVL C00375 V=11.2  //INTO 2ND OB
MOVL C00376 V=11.2
MOVC C00377 V=11.2
MOVC C00378 V=11.2
MOVC C00379 V=11.2
MOVL C00380 V=11.2
MOVC C00381 V=11.2
MOVC C00382 V=11.2
MOVC C00383 V=11.2
MOVL C00384 V=11.2  //END
MOVL C00385 V=33.7  //OUT
SFTOF
MOVJ C00386 VJ=48.75
MOVJ C00387 VJ=48.75
MOVJ C00388 VJ=48.75
MOVJ C00389 VJ=48.75  //OYHER SIDE
MOVL C00390 V=11.2  //INTO
MOVL C00391 V=11.2
MOVC C00392 V=11.2
MOVC C00393 V=11.2
MOVC C00394 V=11.2
MOVC C00395 V=11.2
MOVL C00396 V=11.2
MOVC C00397 V=11.2
MOVC C00398 V=11.2
MOVC C00399 V=11.2
MOVC C00400 V=11.2
MOVL C00401 V=11.2  //END
MOVL C00402 V=11.2  //AWAY
MOVL C00403 V=33.7  //OUT
MOVL C00404 V=65.0  //OVER TO 2ND LEFT
MOVL C00405 V=11.2  //INTO
MOVC C00406 V=11.2
MOVC C00407 V=11.2
MOVC C00408 V=11.2
MOVL C00409 V=11.2
MOVC C00410 V=11.2
MOVC C00411 V=11.2
MOVC C00412 V=11.2
MOVC C00413 V=11.2  //END
MOVL C00414 V=11.2  //AWAY
MOVL C00415 V=33.7  //OUT
MOVJ C00416 VJ=48.75
MOVJ C00417 VJ=48.75
MOVJ C00418 VJ=48.75
MOVJ C00419 VJ=48.75
MOVL C00420 V=65.0  //UP TO FRONT OB
MOVL C00421 V=11.2  //INTO FRONT OB
MOVL C00422 V=11.2
MOVC C00423 V=11.2
MOVC C00424 V=11.2
MOVC C00425 V=11.2
MOVL C00426 V=11.2
MOVC C00427 V=11.2
MOVC C00428 V=11.2
MOVC C00429 V=11.2
MOVL C00430 V=11.2  //END
MOVL C00431 V=11.2
MOVL C00432 V=33.7  //OUT
MOVL C00433 V=33.7  //UP TO BACK OB
MOVL C00434 V=11.2  //INTO BACK OB
MOVL C00435 V=11.2
MOVC C00436 V=11.2
MOVC C00437 V=11.2
MOVC C00438 V=11.2
MOVL C00439 V=11.2
MOVC C00440 V=11.2
MOVC C00441 V=11.2
MOVC C00442 V=11.2
MOVL C00443 V=11.2
MOVL C00444 V=11.2  //END
MOVL C00445 V=11.2  //OUT
MOVL C00446 V=65.0  //AWAY
MOVJ C00447 VJ=48.75
MOVJ C00448 VJ=48.75
MOVJ C00449 VJ=48.75
MOVJ C00450 VJ=48.75  //CENTER
MOVJ C00451 VJ=48.75
MOVL C00452 V=65.0  //UP TO FRONT OB
MOVL C00453 V=11.2  //INTO FRONT OB
MOVL C00454 V=11.2
MOVC C00455 V=11.2
MOVC C00456 V=11.2
MOVC C00457 V=11.2
MOVL C00458 V=11.2
MOVC C00459 V=11.2
MOVC C00460 V=11.2
MOVC C00461 V=11.2
MOVL C00462 V=11.2
MOVL C00463 V=11.2  //END
MOVL C00464 V=33.7  //OUT
MOVL C00465 V=33.7  //UP TO BACK
MOVL C00466 V=11.2  //INTO BACK OB
MOVL C00467 V=11.2
MOVC C00468 V=11.2
MOVC C00469 V=11.2
MOVC C00470 V=11.2
MOVL C00471 V=11.2
MOVC C00472 V=11.2
MOVC C00473 V=11.2
MOVC C00474 V=11.2
MOVL C00475 V=11.2
MOVL C00476 V=11.2  //END
MOVL C00477 V=11.2  //OUT
MOVL C00478 V=65.0  //AWAY
MOVJ C00479 VJ=48.75
MOVJ C00480 VJ=48.75  //CENTER
MOVJ C00481 VJ=48.75  //OUTSIDE
MOVJ C00482 VJ=48.75
MOVJ C00483 VJ=48.75
MOVL C00484 V=65.0  //UP TO OB
SFTON P102
MOVL C00485 V=11.2  //INTO BACK OB
MOVL C00486 V=11.2
MOVC C00487 V=11.2
MOVC C00488 V=11.2
MOVC C00489 V=11.2
MOVL C00490 V=11.2
MOVC C00491 V=11.2
MOVC C00492 V=11.2
MOVC C00493 V=11.2
MOVL C00494 V=11.2
MOVL C00495 V=11.2  //END
SFTOF
MOVL C00496 V=33.7  //OUT
MOVL C00497 V=33.7  //UP TO FRONT OB
SFTON P102
MOVL C00498 V=11.2  //INTO FRONT OB
MOVL C00499 V=11.2  //START
MOVC C00500 V=11.2
MOVC C00501 V=11.2
MOVC C00502 V=11.2
MOVL C00503 V=11.2
MOVC C00504 V=11.2
MOVC C00505 V=11.2
MOVC C00506 V=11.2
MOVL C00507 V=11.2
MOVL C00508 V=11.2  //END
SFTOF
MOVL C00509 V=33.7  //OUT
MOVL C00510 V=65.0  //ABOVE
MOVJ C00511 VJ=48.75
MOVJ C00512 VJ=48.75
MOVJ C00513 VJ=48.75
SFTON P103
MOVL C00514 V=11.2  //INTO
MOVC C00515 V=11.2
MOVC C00516 V=11.2
MOVC C00517 V=11.2
MOVL C00518 V=11.2
MOVC C00519 V=11.2
MOVC C00520 V=11.2
MOVC C00521 V=11.2
MOVC C00522 V=11.2  //END
SFTOF
MOVL C00523 V=11.2  //AWAY
MOVL C00524 V=33.7  //OUT
MOVJ C00525 VJ=48.75
MOVJ C00526 VJ=48.75
MOVJ C00527 VJ=48.75
MOVL C00528 V=65.0  //UP TO
MOVL C00529 V=11.2  //INTO 1
FORMCUT FCF#(1)
MOVL C00530 V=33.7  //OUT
MOVL C00531 V=65.0  //UP TO 2
MOVL C00532 V=11.2  //INTO 2
FORMCUT FCF#(1)
MOVL C00533 V=33.7  //OUT
MOVL C00534 V=65.0  //UP TO 3
MOVL C00535 V=11.2  //INTO 3
FORMCUT FCF#(1)
MOVL C00536 V=33.7  //OUT OF 3
MOVL C00537 V=65.0  //UP TO 4
MOVL C00538 V=11.2  //INTO 4
FORMCUT FCF#(1)
MOVL C00539 V=33.7  //OUT
CALL JOB:SYS_SPINDLE_STOP
MOVJ C00540 VJ=48.75
MOVJ C00541 VJ=48.75
MOVJ C00542 VJ=48.75
MOVJ C00543 VJ=48.75
MOVJ C00544 VJ=48.75  //HOME
CALL JOB:SYS_UNLOCK_GATE
PAUSE
CALL JOB:SYS_FILTERS_STOP
CALL JOB:SYS_UNLOCK_GATE
END
